// TIA Portal V19 export
DATA_BLOCK "DB_Korbumlaeufe"   // DB330
{ S7_Optimized_Access := 'TRUE' }
// stored: AutoNumber false, MemoryReserve 100
   VAR RETAIN
      Korb : Array[1..28] of Struct
         Durchlaeufe : Int;
         max_Durchlaeufe : Int;
         Warnung : Bool;
         max_erreicht : Bool;
      END_STRUCT;
   END_VAR
BEGIN
   Korb[1..13].max_Durchlaeufe := 15;
END_DATA_BLOCK
